SUBAPPLICATION Tuple (* 1 Button, 1 Softkey, 1 Aux *)
  (* Standard: 61499-2 *)
  (* Version 1.0, 2023-02-17, Franz *)
  PACKAGE FBs::Counter::subs::Buttons;
  IMPORT isobus::UT::Q::const::IDs::ID_NULL;
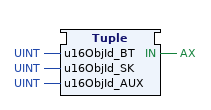
  VAR_INPUT
    u16ObjId_BT : UINT := ID_NULL; (* Object ID Button *)
    u16ObjId_SK : UINT := ID_NULL; (* Object ID SoftKey *)
    u16ObjId_AUX : UINT := ID_NULL; (* Object ID Aux *)
  END_VAR
  PLUGS
    IN : adapter::types::unidirectional::AX;
  END_PLUGS
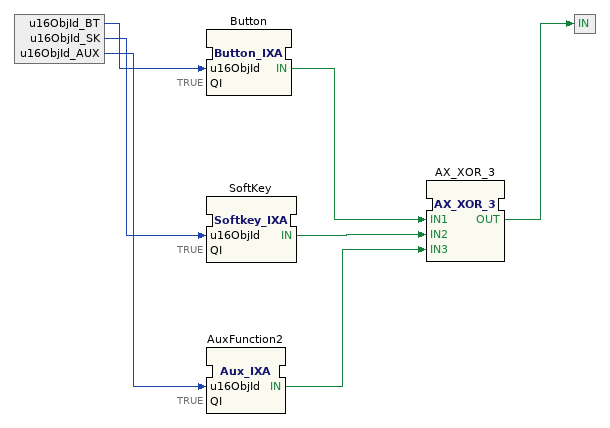
  FBS
    Button : isobus::UT::io::Button::Button_IXA(QI := TRUE);
    SoftKey : isobus::UT::io::Softkey::Softkey_IXA(QI := TRUE);
    AuxFunction2 : isobus::UT::io::Auxiliary::IN::Aux_IXA(QI := TRUE);
    AX_XOR_3 : adapter::booleanOperators::AX_XOR_3;
  END_FBS
  DATA_CONNECTIONS
    u16ObjId_BT TO Button.u16ObjId;
    u16ObjId_SK TO SoftKey.u16ObjId;
    u16ObjId_AUX TO AuxFunction2.u16ObjId;
  END_CONNECTIONS
  ADAPTER_CONNECTIONS
    AX_XOR_3.OUT TO IN;
    Button.IN TO AX_XOR_3.IN1;
    SoftKey.IN TO AX_XOR_3.IN2;
    AuxFunction2.IN TO AX_XOR_3.IN3;
  END_CONNECTIONS
END_SUBAPPLICATION
